// TIA Portal project "RicaII_trabalho_Keslley_versao4" (V18)

(* hardware
DEVICE "S7-1200 station_1"  S7-1200 Station
   slot 0: "Rack_0"  S7-1200 Rack  Rack  V1.0
   slot 1: "PLC_1"  CPU 1214C AC/DC/Rly  6ES7 214-1BE30-0XB0  V2.0
DEVICE "HMI_1"  KTP600 Basic color PN
   slot 0: "HMI_1"  KTP600 Basic color PN  6AV6 647-0AD11-3AX0  12.0.0.0
   slot 1: "HMI_RT_1"  KTP600 Basic color PN  6AV6 647-0AD11-3AX0  12.0.0.0
   slot 5: "HMI_1.IE_CP_1"  PROFINET Interface  12.0.0.0
      slot 1: "PROFINET Interface_1"  PROFINET Interface
         slot 1: "Port_1"  Port
DEVICE "GSD device_1"  GSD.Device.PN
   slot 0: "Rack"  Rack  V1.0
   slot 0: "nl51ndpl"  NL 51N-DPL  NL 51N-DPL
      slot 0: "Useable Module"  Useable Module
      slot 1: "Interface 1"  Interface 1
         slot 1: "Interface 1 - Port1"  Interface 1 - Port1
      slot 1: "NL51N (PROFIBUS-DP)_1"  NL51N (PROFIBUS-DP)  MasterOrderNumber
         slot 0: "Empty module"  Empty module
      slot 76: "1734-APB_1"  1734-APB  SlaveOrderNumber
         slot 0: "1734-IR2"  1734-IR2   ModuleOrderNumber
*)

// ===== PLC "PLC_1"  CPU 1214C AC/DC/Rly =====

VAR_GLOBAL   // PLC tag table "Remota"
   "AI1_TEMP" AT %MW5 : Word;
   "AO1_OXIGENIO" AT %MW10 : Word;
   "AO2_GAS" AT %MW12 : Word;
   "LED_ON_OFF" AT %MW14 : Word;
   "AI1_TEMP_R" AT %MD1 : Real;
   "AI1_TEMP_I" AT %MW16 : Int;
   "AO1_OXIGENIO_REAL" AT %MD22 : Real;
   "AO2_GAS_REAL" AT %MD24 : Real;
   "AO1_OXIGENIO_INT" AT %MW28 : Int;
   "AO2_GAS_INT" AT %MW32 : Int;
   "ALARMES" AT %MW8 : Word;   // Bit0: botão alarme; Bit2: on_off; Bit3: conexão nl51
END_VAR

VAR_GLOBAL   // PLC tag table "NL51"
   "NL51_SETPOINT_1600" AT %MW78 : Word;
   "NL51_SETPOINT_N" AT %MD74 : Real;
   "NL51_SETPOINT" AT %IW68 : Word;
   "NL51_PLC_ACK" AT %MW72 : Word;
   "NL51_PLC_ALARM" AT %MW70 : Word;
   "NL51_SETPOINT_I" AT %MW80 : Int;
   "NL51_SETPOINT_R" AT %MD38 : Real;
END_VAR

VAR_GLOBAL   // PLC tag table "Modbus"
   "System_Byte" AT %MB1 : Byte;
   "FirstScan" AT %M1.0 : Bool;
   "DiagStatusUpdate" AT %M1.1 : Bool;
   "AlwaysTRUE" AT %M1.2 : Bool;
   "AlwaysFALSE" AT %M1.3 : Bool;
   "Clock_Byte" AT %MB0 : Byte;
   "Clock_10Hz" AT %M0.0 : Bool;
   "Clock_5Hz" AT %M0.1 : Bool;
   "Clock_2.5Hz" AT %M0.2 : Bool;
   "Clock_2Hz" AT %M0.3 : Bool;
   "Clock_1.25Hz" AT %M0.4 : Bool;
   "Clock_1Hz" AT %M0.5 : Bool;
   "Clock_0.625Hz" AT %M0.6 : Bool;
   "Clock_0.5Hz" AT %M0.7 : Bool;
END_VAR

VAR_GLOBAL   // PLC tag table "PID"
   "PID_SETPOINT_PERCENTUAL" AT %MD42 : Real;
   "PID_SETPOINT_N" AT %MD46 : Real;
   "PID_IN_N" AT %MD50 : Real;
   "PID_IN_PERCENTUAL" AT %MD54 : Real;
END_VAR

DATA_BLOCK "Global DB"   // DB1
{ S7_Optimized_Access := 'FALSE' }
VERSION : 0.1
   VAR
      MB_ConnectID : Word := 1;
      MB_Mode : Byte := 0;
      MB_DataAddr : Word := 40001;
      MB_Datalen : Word := 5;
      MB_Data : Array[1..5] of Word;
      MB_Done : Bool;
      MB_Busy : Bool;
      MB_Error : Bool;
      MB_Status : Word;
   END_VAR
BEGIN
END_DATA_BLOCK

DATA_BLOCK "HMI_DATA"   // DB3
{ S7_Optimized_Access := 'TRUE' }
VERSION : 0.1
   VAR
      HMI_LED_ON_OFF : Bool;
   END_VAR
BEGIN
END_DATA_BLOCK

ORGANIZATION_BLOCK "Main"   // OB1, LAD, ProgramCycle
TITLE = "Main Program Sweep (Cycle)"
{ S7_Optimized_Access := 'TRUE' }
VERSION : 0.1
BEGIN

REGION Network 1
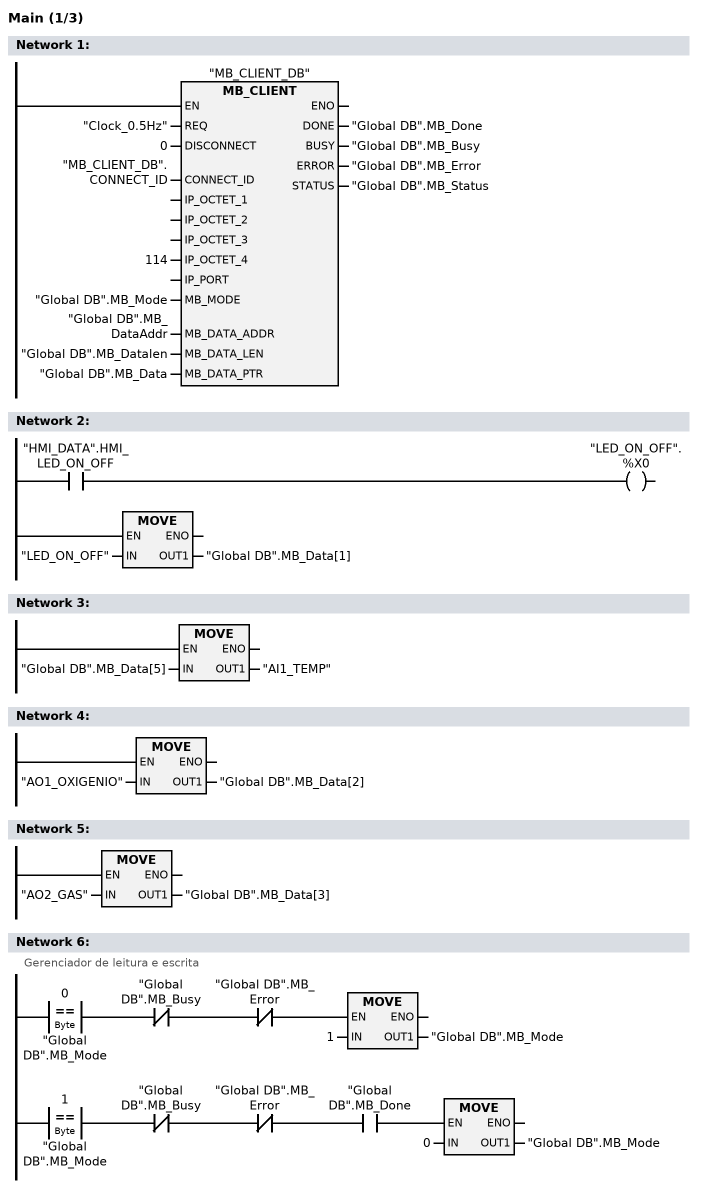
   "MB_CLIENT_DB"(REQ := "Clock_0.5Hz",   // MB_CLIENT
                  DISCONNECT := 0,
                  CONNECT_ID := "MB_CLIENT_DB".CONNECT_ID,
                  IP_OCTET_4 := 114,
                  MB_MODE := "Global DB".MB_Mode,
                  MB_DATA_ADDR := "Global DB".MB_DataAddr,
                  MB_DATA_LEN := "Global DB".MB_Datalen,
                  MB_DATA_PTR := "Global DB".MB_Data,
                  DONE => "Global DB".MB_Done,
                  BUSY => "Global DB".MB_Busy,
                  ERROR => "Global DB".MB_Error,
                  STATUS => "Global DB".MB_Status);
END_REGION

REGION Network 2
   RUNG wire#powerrail
      Contact( "HMI_DATA".HMI_LED_ON_OFF )
      Coil( "LED_ON_OFF".%X0 )
   END_RUNG
   RUNG wire#powerrail
      { S7_GenerateENO := "TRUE" } Move(in := "LED_ON_OFF", out1 => "Global DB".MB_Data[1])
   END_RUNG
   // the same network as SCL:
   "LED_ON_OFF".%X0 := "HMI_DATA".HMI_LED_ON_OFF;
   "Global DB".MB_Data[1] := "LED_ON_OFF";
END_REGION

REGION Network 3
   RUNG wire#powerrail
      { S7_GenerateENO := "TRUE" } Move(in := "Global DB".MB_Data[5], out1 => "AI1_TEMP")
   END_RUNG
   // the same network as SCL:
   "AI1_TEMP" := "Global DB".MB_Data[5];
END_REGION

REGION Network 4
   RUNG wire#powerrail
      { S7_GenerateENO := "TRUE" } Move(in := "AO1_OXIGENIO", out1 => "Global DB".MB_Data[2])
   END_RUNG
   // the same network as SCL:
   "Global DB".MB_Data[2] := "AO1_OXIGENIO";
END_REGION

REGION Network 5
   RUNG wire#powerrail
      { S7_GenerateENO := "TRUE" } Move(in := "AO2_GAS", out1 => "Global DB".MB_Data[3])
   END_RUNG
   // the same network as SCL:
   "Global DB".MB_Data[3] := "AO2_GAS";
END_REGION

REGION Network 6
   // Gerenciador de leitura e escrita
   RUNG wire#powerrail
      { S7_Templates := "SrcType := Byte" } EQ_Contact(in1 := 0, in2 := "Global DB".MB_Mode)
      I_Contact( "Global DB".MB_Busy )
      I_Contact( "Global DB".MB_Error )
      { S7_GenerateENO := "TRUE" } Move(in := 1, out1 => "Global DB".MB_Mode)
   END_RUNG
   RUNG wire#powerrail
      { S7_Templates := "SrcType := Byte" } EQ_Contact(in1 := 1, in2 := "Global DB".MB_Mode)
      I_Contact( "Global DB".MB_Busy )
      I_Contact( "Global DB".MB_Error )
      Contact( "Global DB".MB_Done )
      { S7_GenerateENO := "TRUE" } Move(in := 0, out1 => "Global DB".MB_Mode)
   END_RUNG
   // the same network as SCL:
   IF (0 = "Global DB".MB_Mode) AND NOT "Global DB".MB_Busy AND NOT "Global DB".MB_Error THEN
       "Global DB".MB_Mode := 1;
   END_IF;
   IF (1 = "Global DB".MB_Mode) AND NOT "Global DB".MB_Busy AND NOT "Global DB".MB_Error AND "Global DB".MB_Done THEN
       "Global DB".MB_Mode := 0;
   END_IF;
END_REGION

REGION Network 7
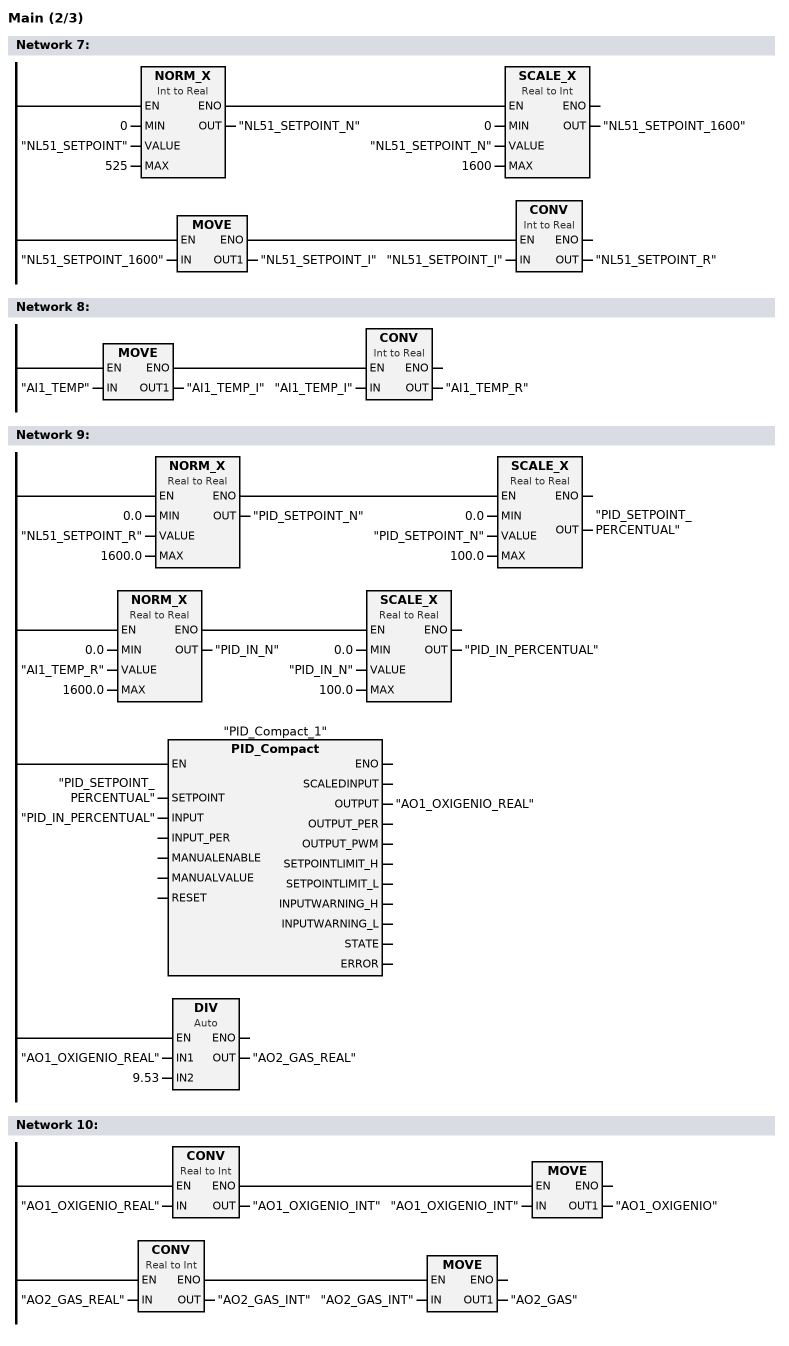
   RUNG wire#powerrail
      { S7_Templates := "[SrcType := Int, DestType := Real]"; S7_GenerateENO := "TRUE" } Normalize(min := 0, value := "NL51_SETPOINT", max := 525, out => "NL51_SETPOINT_N")
      { S7_Templates := "[SrcType := Real, DestType := Int]"; S7_GenerateENO := "TRUE" } Scale(min := 0, value := "NL51_SETPOINT_N", max := 1600, out => "NL51_SETPOINT_1600")
   END_RUNG
   RUNG wire#powerrail
      { S7_GenerateENO := "TRUE" } Move(in := "NL51_SETPOINT_1600", out1 => "NL51_SETPOINT_I")
      { S7_Templates := "[SrcType := Int, DestType := Real]"; S7_GenerateENO := "TRUE" } Convert(in := "NL51_SETPOINT_I", out => "NL51_SETPOINT_R")
   END_RUNG
   // the same network as SCL:
   // ENO of a box is taken as its EN; it also drops when the box reports an error
   "NL51_SETPOINT_N" := NORM_X(MIN := 0, VALUE := "NL51_SETPOINT", MAX := 525);
   "NL51_SETPOINT_1600" := SCALE_X(MIN := 0, VALUE := "NL51_SETPOINT_N", MAX := 1600);
   "NL51_SETPOINT_I" := "NL51_SETPOINT_1600";
   "NL51_SETPOINT_R" := INT_TO_REAL("NL51_SETPOINT_I");
END_REGION

REGION Network 8
   RUNG wire#powerrail
      { S7_GenerateENO := "TRUE" } Move(in := "AI1_TEMP", out1 => "AI1_TEMP_I")
      { S7_Templates := "[SrcType := Int, DestType := Real]"; S7_GenerateENO := "TRUE" } Convert(in := "AI1_TEMP_I", out => "AI1_TEMP_R")
   END_RUNG
   // the same network as SCL:
   // ENO of a box is taken as its EN; it also drops when the box reports an error
   "AI1_TEMP_I" := "AI1_TEMP";
   "AI1_TEMP_R" := INT_TO_REAL("AI1_TEMP_I");
END_REGION

REGION Network 9
   // ENO of a box is taken as its EN; it also drops when the box reports an error
   "PID_SETPOINT_N" := NORM_X(MIN := 0.0, VALUE := "NL51_SETPOINT_R", MAX := 1600.0);
   "PID_SETPOINT_PERCENTUAL" := SCALE_X(MIN := 0.0, VALUE := "PID_SETPOINT_N", MAX := 100.0);
   "PID_IN_N" := NORM_X(MIN := 0.0, VALUE := "AI1_TEMP_R", MAX := 1600.0);
   "PID_IN_PERCENTUAL" := SCALE_X(MIN := 0.0, VALUE := "PID_IN_N", MAX := 100.0);
   "PID_Compact_1"(Setpoint := "PID_SETPOINT_PERCENTUAL",   // PID_Compact
                   Input := "PID_IN_PERCENTUAL",
                   Output => "AO1_OXIGENIO_REAL");
   "AO2_GAS_REAL" := "AO1_OXIGENIO_REAL" / 9.53;
END_REGION

REGION Network 10
   RUNG wire#powerrail
      { S7_Templates := "[SrcType := Real, DestType := Int]"; S7_GenerateENO := "TRUE" } Convert(in := "AO1_OXIGENIO_REAL", out => "AO1_OXIGENIO_INT")
      { S7_GenerateENO := "TRUE" } Move(in := "AO1_OXIGENIO_INT", out1 => "AO1_OXIGENIO")
   END_RUNG
   RUNG wire#powerrail
      { S7_Templates := "[SrcType := Real, DestType := Int]"; S7_GenerateENO := "TRUE" } Convert(in := "AO2_GAS_REAL", out => "AO2_GAS_INT")
      { S7_GenerateENO := "TRUE" } Move(in := "AO2_GAS_INT", out1 => "AO2_GAS")
   END_RUNG
   // the same network as SCL:
   // ENO of a box is taken as its EN; it also drops when the box reports an error
   "AO1_OXIGENIO_INT" := REAL_TO_INT("AO1_OXIGENIO_REAL");
   "AO1_OXIGENIO" := "AO1_OXIGENIO_INT";
   "AO2_GAS_INT" := REAL_TO_INT("AO2_GAS_REAL");
   "AO2_GAS" := "AO2_GAS_INT";
END_REGION

REGION Network 11: Alarmes
   // Bit0: botão alarme; Bit2: on_off; Bit1 e 3: conexão nl51; Bit4: conexão modbus
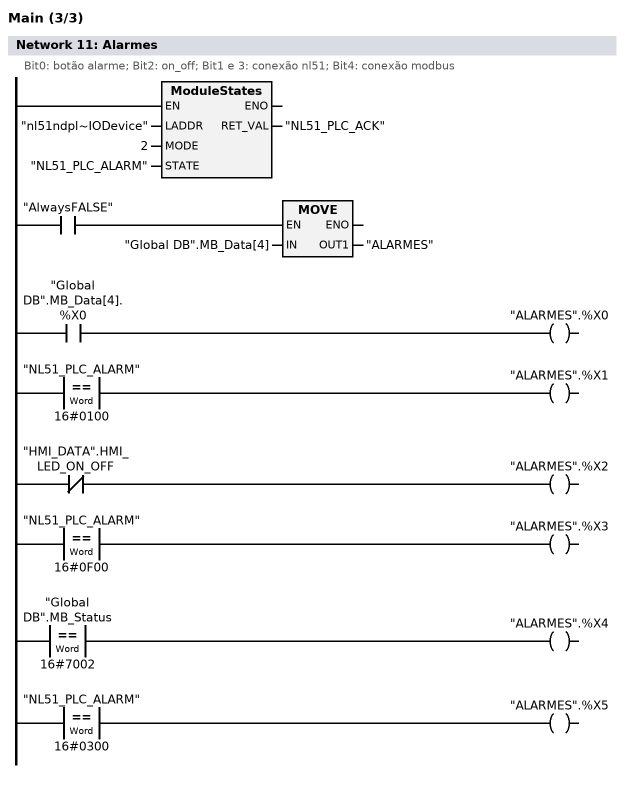
   // no SCL statement known for ModuleStates: written as a call
   "NL51_PLC_ACK" := ModuleStates(LADDR := "nl51ndpl~IODevice", MODE := 2, STATE := "NL51_PLC_ALARM");
   IF "AlwaysFALSE" THEN "ALARMES" := "Global DB".MB_Data[4]; END_IF;
   "ALARMES".%X0 := "Global DB".MB_Data[4].%X0;
   "ALARMES".%X1 := "NL51_PLC_ALARM" = 16#0100;
   "ALARMES".%X2 := NOT "HMI_DATA".HMI_LED_ON_OFF;
   "ALARMES".%X3 := "NL51_PLC_ALARM" = 16#0F00;
   "ALARMES".%X4 := "Global DB".MB_Status = 16#7002;
   "ALARMES".%X5 := "NL51_PLC_ALARM" = 16#0300;
END_REGION
END_ORGANIZATION_BLOCK

(* ===== HMI "HMI_RT_1" =====
system functions are stored by id; their names below are inferred from use
connection "HMI_Connection_1": ETHERNET, SMART_S7_1200_OMS

HMI tags "Default tag table"
   "HMI_AI1_TEMP" : Word = PLC AI1_TEMP AT %MW5, 1 s
   "HMI_LED_ON_OFF" : Bool = PLC HMI_DATA.HMI_LED_ON_OFF, 1 s
   "HMI_AO1_OXIGENIO" : Word = PLC AO1_OXIGENIO AT %MW10, 1 s
   "HMI_AO2_GAS" : Word = PLC AO2_GAS AT %MW12, 1 s
   "Global DB_MB_Mode" : Byte = PLC "Global DB".MB_Mode AT %DB1.DBB2, 1 s
   "IHM_ALM" : Word = PLC ALARMES AT %MW8, 1 s
   "IHM_ALM_NL51" : Word = PLC NL51_PLC_ALARM AT %MW70, 1 s
   "IHM_ACK_NL51" : Word = PLC NL51_PLC_ACK AT %MW72, 1 s
   "IHM_SETPOINT_PID" : Real = PLC NL51_SETPOINT_R AT %MD38, 1 s

discrete alarms
   1: 'Botão de Alarme pressionado!', class Warnings, trigger "IHM_ALM" bit 0
   2: 'Erro em um canal do Slave NL51 (setpoint)', class Errors, trigger "IHM_ALM" bit 1
   5: 'Remota modbusTCP está desligada. (valvulas desabilitadas)', class Warnings, trigger "IHM_ALM" bit 2
   3: 'O Slave NL51 (setpoint) não está respondendo.', class Errors, trigger "IHM_ALM" bit 3
   6: 'Erro na Remota modbusTCP. (Verifique a conexão)', class Errors, trigger "IHM_ALM" bit 4
   4: 'O Slave NL51 (setpoint) foi desconectado.', class Errors, trigger "IHM_ALM" bit 5

analog alarms
   10: 'Temperatura acima de 1400ºC', class Errors, trigger "HMI_AI1_TEMP"
   11: 'Temperatura abaixo de 200ºC', class Errors, trigger "HMI_AI1_TEMP"

Template "Template_1" 320x240
   Button "Exit" at 278,208 size 42x30; TextOff 'Exit'; PictureOff "ExitRuntime_KTP600_Basic_color_PN"; PictureOn "ExitRuntime_KTP600_Basic_color_PN"
      on Release: StopRuntime(0)
   Button "Template_Button" at 231,208 size 42x30; TextOff 'TAlarm'; TextList "T"
      on Press: ActivateScreen("TAlarm", 0)
   Button "Template_Button_1" at 183,208 size 42x30; TextOff 'TG'
      on Press: ActivateScreen("TGRAPH_TEMP_ESP", 0)
   Button "Template_Button_2" at 90,208 size 42x30; TextOff 'AO'
      on Press: ActivateScreen("TANALOG_OUT_BARRA", 0)
   Button "Alarms" at 45,208 size 42x30; TextOff 'TD'; TextOn 'Alarms'; PictureOff "AlarmDisplay_KTP600_Basic_color_PN"; PictureOn "AlarmDisplay_KTP600_Basic_color_PN"
      on Press: ActivateScreen("TDIGITAL", 0)
   Button "Start screen" at 0,208 size 42x30; TextOff 'Start screen'; PictureOff "NavigateHome_KTP600_Basic_color_PN"; PictureOn "NavigateHome_KTP600_Basic_color_PN"
      on Release: ActivateScreen("Root screen", 0)
   Button "Template_Button_3" at 136,208 size 42x30; TextOff 'AI'
      on Press: ActivateScreen("TANALOG_IN", 0)

screen "Root screen" 320x240, template "Template_1"
   TextField "HmiScreenItemData" at 0,0 size 320x48; Text 'MONITORAMENTO DO FORNO DE FUSÃO DE VIDROS'
   GraphicView "Graphic view_1" at 34,42 size 259x156; Picture "imagem forno"

screen "TDIGITAL" 320x240, template "Template_1"
   Circle "Circle_1" at 17,64 size 48x48
      Appearance <- "HMI_LED_ON_OFF"
   Button "Button_1" at 4,124 size 77x32; TextOff 'ON/OFF'
      on Press: InvertBit("HMI_LED_ON_OFF")
   TextField "Text field_1" at 20,12 size 284x16; Text 'Painel de Inicialização da Remota Modbus TCP'
   TextField "Text field_2" at 96,64 size 221x35; Text 'Para inicializar o sistema, pressione o botão "ON/OFF" e aguarde até que acenda o LED verde da tela e o LED vermelho na remota.'
   TextField "Text field_3" at 99,123 size 218x46; Text 'Para desligar o sistema, pressione o botão "ON/OFF" e aguarde até que acenda o LED vermelho da tela e que o LED vermelho da remota se apague.'

screen "TANALOG_OUT_BARRA" 320x240, template "Template_1"
   Button "Back" at 278,0 size 42x30; TextOff 'Back'
      on Release: ActivateScreen("Root screen", 0)
   Bar "Bar_1" at 29,62 size 68x95; MinimumValue 0; MaximumValue 100
      ProcessValue <- "HMI_AO1_OXIGENIO"
   IOField "I/O field_1" at 44,163 size 39x20; FormatPattern 9999
      ProcessValue <- "HMI_AO1_OXIGENIO"
   Bar "Bar_2" at 129,62 size 72x95; MinimumValue 0; MaximumValue 100
      ProcessValue <- "HMI_AO2_GAS"
   IOField "I/O field_2" at 143,163 size 39x20; FormatPattern 9999
      ProcessValue <- "HMI_AO2_GAS"
   TextField "Text field_2" at 35,39 size 62x18; Text 'OXIGÊNIO'
   TextField "Text field_3" at 18,0 size 257x25; Text 'Abertura das Valvulas (%)'
   TextField "Text field_1" at 151,39 size 28x18; Text 'GÁS'
   Button "Button_2" at 264,39 size 56x35; TextOff 'GRÁFICO PID'
      on Click: ActivateScreen("TANALOG_OUT_GRAFICOPID", 0)

screen "TAlarm" 320x240, template "Template_1"
   AlarmView "Alarm view_1" at 0,30 size 320x172
   Button "Button_1" at 104,170 size 96x32; TextOff 'Clear'
      on Press: function_e14cd482(0)
   TextField "Text field_1" at 60,2 size 191x25; Text 'Alarmes do Sistema'

screen "TANALOG_IN" 320x240, template "Template_1"
   Bar "Bar_1" at 118,60 size 80x120; MinimumValue 0; MaximumValue 1600
      ProcessValue <- "HMI_AI1_TEMP"
   Button "Back" at 272,1 size 48x25; TextOn 'Back'; TextOff 'Back'
      on Release: ActivateScreen("Root screen", 0)
   IOField "I/O field_1" at 138,183 size 44x20; FormatPattern 9999
      ProcessValue <- "HMI_AI1_TEMP"
   TextField "Text field_1" at 104,28 size 85x25; Text 'TEMP S1'
   TextField "Text field_3" at 49,5 size 224x48; Text 'Sensor de Temperatura do Forno'

screen "TGRAPH_TEMP_ESP" 320x240, template "Template_1"
   TextField "HmiScreenItemData" at 32,90 size 256x17; Text 'TGRAPH'
   TrendView "Trend view_1" at 7,26 size 302x151
   IOField "I/O field_1" at 201,180 size 49x25; FormatPattern 99999
      ProcessValue <- "HMI_AI1_TEMP"
   TextField "Text field_1" at 58,0 size 204x23; Text 'Gráfico de Temperatura'
   TextField "Text field_2" at 85,186 size 104x13; Text 'Valor em tempo real'
   TextField "Text field_3" at 27,96 size 30x24; Text 'Temp (ºC)'

screen "TANALOG_OUT_GRAFICOPID" 320x240, template "Template_1"
   Button "Back" at 286,0 size 34x18; TextOn 'Back'; TextOff 'Back'
      on Release: ActivateScreen("Root screen", 0)
   TextField "Text field_3" at 97,0 size 130x48; Text 'Abertura das Válvulas'
   TrendView "Trend view_1" at 3,73 size 283x102
   Button "Button_1" at 262,29 size 58x30; TextOff 'GRÁFICO BARRA'
      on Click: ActivateScreen("TANALOG_OUT_BARRA", 0)
   IOField "I/O field_1" at 185,183 size 51x19; FormatPattern s999999999.999
      ProcessValue <- "IHM_SETPOINT_PID"
   TextField "Text field_2" at 76,179 size 109x24; Text 'Setpoint temperatura (0º - 1600º)'
   TextField "Text field_1" at 2,100 size 35x22; Text '% válvulas'
   TextField "Text field_5" at 291,100 size 27x22; Text 'temp média'
   TextField "Text field_6" at 283,151 size 35x12; Text 'Setpoint'
   TextField "Text field_7" at 283,158 size 25x12; Text 'Temp'
   TextField "Text field_8" at 283,166 size 17x12; Text 'Gás'
   TextField "Text field_9" at 283,174 size 13x12; Text 'O2'
*)